// TIA Portal project "Project1" (V17)

(* hardware
DEVICE "S7-1200 station_1"  S7-1200 Station
   slot 0: "Rack_0"  S7-1200 Rack  Rack  V1.0
   slot 1: "PLC_1"  CPU 1215C AC/DC/Rly  6ES7 215-1BG40-0XB0  V4.5
*)

// ===== PLC "PLC_1"  CPU 1215C AC/DC/Rly =====

VAR_GLOBAL   // PLC tag table "input"
   "start" AT %I0.0 : Bool;
   "stop" AT %I0.1 : Bool;
   "cảm biến 1" AT %I0.2 : Bool;
   "cảm biến 2" AT %I0.3 : Bool;
   "cảm biến 3" AT %I0.4 : Bool;
   "cảm biến 4" AT %I0.5 : Bool;
   "cảm biến 5" AT %I0.6 : Bool;
   "auto" AT %I0.7 : Bool;
   "manual" AT %I1.0 : Bool;
   "emc" AT %I1.1 : Bool;
   "process1" AT %I1.2 : Bool;
   "process2" AT %I1.3 : Bool;
   "process3" AT %I1.4 : Bool;
END_VAR

VAR_GLOBAL   // PLC tag table "bit trung gian"
   "Tag_3" AT %M0.0 : Bool;
   "cam bien 1" AT %M0.1 : Bool;
   "hàng đỏ" AT %M1.0 : Bool;
   "hàng xanh lá" AT %M1.1 : Bool;
   "hàng xanh dương" AT %M1.2 : Bool;
   "hàng NG" AT %M1.3 : Bool;
   "cam bien 2" AT %M0.2 : Bool;
   "cảm bien 3" AT %M0.3 : Bool;
   "cam bien 4" AT %M0.4 : Bool;
   "cam bien 5" AT %M0.5 : Bool;
   "bit nho hang NG" AT %M0.6 : Bool;
   "bit nho van day 1" AT %M2.0 : Bool;
   "bit nho van day 2" AT %M2.1 : Bool;
   "Tag_4" AT %M2.2 : Bool;
   "Tag_5" AT %M2.3 : Bool;
   "bit nho van SP do" AT %M2.5 : Bool;
   "bit nho van SP xanh la" AT %M2.6 : Bool;
   "bit nho van sp xanh duong" AT %M2.7 : Bool;
   "bit nho van SP do 2" AT %M2.4 : Bool;
   "reset" AT %M3.0 : Bool;
   "bit nho bang tai" AT %M4.0 : Bool;
   "bit nho van xoay" AT %M4.1 : Bool;
   "bit nho van kep" AT %M4.2 : Bool;
   "bit nho van SP do 3" AT %M4.3 : Bool;
   "bit nho van xanh la 2" AT %M4.4 : Bool;
END_VAR

VAR_GLOBAL   // PLC tag table "bit output"
   "băng tải" AT %Q0.0 : Bool;
   "van sp đỏ" AT %Q0.1 : Bool;
   "Đèn xanh" AT %Q0.7 : Bool;
   "Đèn đỏ" AT %Q1.0 : Bool;
   "van xoay" AT %Q0.4 : Bool;
   "van đẩy tay gắp" AT %Q0.5 : Bool;
   "van kẹp tay gắp" AT %Q0.6 : Bool;
   "van sp xanh lá" AT %Q0.2 : Bool;
   "van sp xanh dương" AT %Q0.3 : Bool;
   "Đèn vàng" AT %Q1.1 : Bool;
END_VAR

DATA_BLOCK "DB1"   // DB1
{ S7_Optimized_Access := 'TRUE' }
VERSION : 0.1
   VAR
      disconnect : Bool;
      connect : TCON_IP_v4;
      error : Bool;
      h_reg : Array[0..50] of Int;
      status : Word;
   END_VAR
BEGIN
   connect.InterfaceId := 64;
   connect.ID := 1;
   connect.ConnectionType := 11;
   connect.LocalPort := 502;
   h_reg[16] := 0;
END_DATA_BLOCK

// folder: System blocks/Program resources

DATA_BLOCK "counter start"   // DB3
{ S7_Optimized_Access := 'TRUE' }
AUTHOR : Simatic
FAMILY : IEC
NAME : CNTR
VERSION : 1.0
// stored: InstanceOfName IEC_COUNTER
"IEC_COUNTER"
BEGIN
END_DATA_BLOCK

DATA_BLOCK "counter stop"   // DB4
{ S7_Optimized_Access := 'TRUE' }
AUTHOR : Simatic
FAMILY : IEC
NAME : CNTR
VERSION : 1.0
// stored: InstanceOfName IEC_COUNTER
"IEC_COUNTER"
BEGIN
END_DATA_BLOCK

DATA_BLOCK "T1"   // DB5
{ S7_Optimized_Access := 'TRUE' }
AUTHOR : Simatic
FAMILY : IEC
NAME : IEC_TMR
VERSION : 1.0
// stored: InstanceOfName IEC_TIMER
"IEC_TIMER"
BEGIN
END_DATA_BLOCK

DATA_BLOCK "timer hang xanh duong"   // DB6
{ S7_Optimized_Access := 'TRUE' }
AUTHOR : Simatic
FAMILY : IEC
NAME : IEC_TMR
VERSION : 1.0
// stored: InstanceOfName IEC_TIMER
"IEC_TIMER"
BEGIN
END_DATA_BLOCK

DATA_BLOCK "Counter dem hang xanh duong"   // DB7
{ S7_Optimized_Access := 'TRUE' }
AUTHOR : Simatic
FAMILY : IEC
NAME : CNTR
VERSION : 1.0
// stored: InstanceOfName IEC_COUNTER
"IEC_COUNTER"
BEGIN
END_DATA_BLOCK

DATA_BLOCK "xanh duong"   // DB8
{ S7_Optimized_Access := 'TRUE' }
AUTHOR : Simatic
FAMILY : IEC
NAME : CNTR
VERSION : 1.0
// stored: InstanceOfName IEC_COUNTER
"IEC_COUNTER"
BEGIN
END_DATA_BLOCK

DATA_BLOCK "đỏ"   // DB9
{ S7_Optimized_Access := 'TRUE' }
AUTHOR : Simatic
FAMILY : IEC
NAME : CNTR
VERSION : 1.0
// stored: InstanceOfName IEC_COUNTER
"IEC_COUNTER"
BEGIN
END_DATA_BLOCK

DATA_BLOCK "Timer hang do"   // DB10
{ S7_Optimized_Access := 'TRUE' }
AUTHOR : Simatic
FAMILY : IEC
NAME : IEC_TMR
VERSION : 1.0
// stored: InstanceOfName IEC_TIMER
"IEC_TIMER"
BEGIN
END_DATA_BLOCK

DATA_BLOCK "Counter dem hang do"   // DB11
{ S7_Optimized_Access := 'TRUE' }
AUTHOR : Simatic
FAMILY : IEC
NAME : CNTR
VERSION : 1.0
// stored: InstanceOfName IEC_COUNTER
"IEC_COUNTER"
BEGIN
END_DATA_BLOCK

DATA_BLOCK "xanh la cay"   // DB12
{ S7_Optimized_Access := 'TRUE' }
AUTHOR : Simatic
FAMILY : IEC
NAME : CNTR
VERSION : 1.0
// stored: InstanceOfName IEC_COUNTER
"IEC_COUNTER"
BEGIN
END_DATA_BLOCK

DATA_BLOCK "Timer xanh la cay"   // DB13
{ S7_Optimized_Access := 'TRUE' }
AUTHOR : Simatic
FAMILY : IEC
NAME : IEC_TMR
VERSION : 1.0
// stored: InstanceOfName IEC_TIMER
"IEC_TIMER"
BEGIN
END_DATA_BLOCK

DATA_BLOCK "Counter dem xanh la cay"   // DB14
{ S7_Optimized_Access := 'TRUE' }
AUTHOR : Simatic
FAMILY : IEC
NAME : CNTR
VERSION : 1.0
// stored: InstanceOfName IEC_COUNTER
"IEC_COUNTER"
BEGIN
END_DATA_BLOCK

DATA_BLOCK "IEC_Counter_0_DB"   // DB15
{ S7_Optimized_Access := 'TRUE' }
AUTHOR : Simatic
FAMILY : IEC
NAME : CNTR
VERSION : 1.0
// stored: InstanceOfName IEC_COUNTER
"IEC_COUNTER"
BEGIN
END_DATA_BLOCK

DATA_BLOCK "bao full do"   // DB16
{ S7_Optimized_Access := 'TRUE' }
AUTHOR : Simatic
FAMILY : IEC
NAME : CNTR
VERSION : 1.0
// stored: InstanceOfName IEC_COUNTER
"IEC_COUNTER"
BEGIN
END_DATA_BLOCK

DATA_BLOCK "bao full xanh la"   // DB17
{ S7_Optimized_Access := 'TRUE' }
AUTHOR : Simatic
FAMILY : IEC
NAME : CNTR
VERSION : 1.0
// stored: InstanceOfName IEC_COUNTER
"IEC_COUNTER"
BEGIN
END_DATA_BLOCK

DATA_BLOCK "bao ful xanh duong"   // DB18
{ S7_Optimized_Access := 'TRUE' }
AUTHOR : Simatic
FAMILY : IEC
NAME : CNTR
VERSION : 1.0
// stored: InstanceOfName IEC_COUNTER
"IEC_COUNTER"
BEGIN
END_DATA_BLOCK

DATA_BLOCK "hang NG"   // DB19
{ S7_Optimized_Access := 'TRUE' }
AUTHOR : Simatic
FAMILY : IEC
NAME : CNTR
VERSION : 1.0
// stored: InstanceOfName IEC_COUNTER
"IEC_COUNTER"
BEGIN
END_DATA_BLOCK

DATA_BLOCK "counter dem hang NG"   // DB20
{ S7_Optimized_Access := 'TRUE' }
AUTHOR : Simatic
FAMILY : IEC
NAME : CNTR
VERSION : 1.0
// stored: InstanceOfName IEC_COUNTER
"IEC_COUNTER"
BEGIN
END_DATA_BLOCK

DATA_BLOCK "bao full NG"   // DB21
{ S7_Optimized_Access := 'TRUE' }
AUTHOR : Simatic
FAMILY : IEC
NAME : CNTR
VERSION : 1.0
// stored: InstanceOfName IEC_COUNTER
"IEC_COUNTER"
BEGIN
END_DATA_BLOCK

DATA_BLOCK "counter cb 1"   // DB22
{ S7_Optimized_Access := 'TRUE' }
AUTHOR : Simatic
FAMILY : IEC
NAME : CNTR
VERSION : 1.0
// stored: InstanceOfName IEC_COUNTER
"IEC_COUNTER"
BEGIN
END_DATA_BLOCK

DATA_BLOCK "T2"   // DB23
{ S7_Optimized_Access := 'TRUE' }
AUTHOR : Simatic
FAMILY : IEC
NAME : IEC_TMR
VERSION : 1.0
// stored: InstanceOfName IEC_TIMER
"IEC_TIMER"
BEGIN
END_DATA_BLOCK

DATA_BLOCK "chay bang tai"   // DB24
{ S7_Optimized_Access := 'TRUE' }
AUTHOR : Simatic
FAMILY : IEC
NAME : CNTR
VERSION : 1.0
// stored: InstanceOfName IEC_COUNTER
"IEC_COUNTER"
BEGIN
END_DATA_BLOCK

DATA_BLOCK "IEC_Counter_0_DB_1"   // DB25
{ S7_Optimized_Access := 'TRUE' }
AUTHOR : Simatic
FAMILY : IEC
NAME : CNTR
VERSION : 1.0
// stored: InstanceOfName IEC_COUNTER
"IEC_COUNTER"
BEGIN
END_DATA_BLOCK

DATA_BLOCK "IEC_Counter_0_DB_2"   // DB26
{ S7_Optimized_Access := 'TRUE' }
AUTHOR : Simatic
FAMILY : IEC
NAME : CNTR
VERSION : 1.0
// stored: InstanceOfName IEC_COUNTER
"IEC_COUNTER"
BEGIN
END_DATA_BLOCK

DATA_BLOCK "IEC_Counter_0_DB_3"   // DB27
{ S7_Optimized_Access := 'TRUE' }
AUTHOR : Simatic
FAMILY : IEC
NAME : CNTR
VERSION : 1.0
// stored: InstanceOfName IEC_COUNTER
"IEC_COUNTER"
BEGIN
END_DATA_BLOCK

// folder: (top level)

FUNCTION "ouput" : Void   // FC1, LAD
{ S7_Optimized_Access := 'TRUE' }
VERSION : 0.1
BEGIN

REGION Network 1
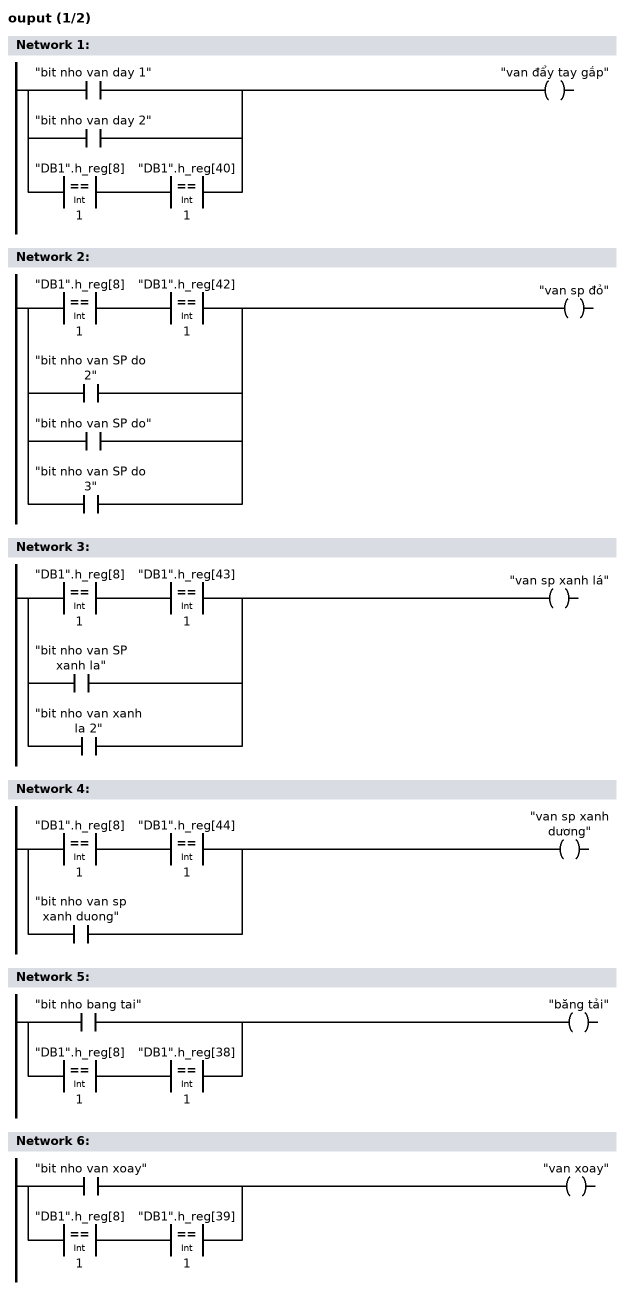
   RUNG wire#powerrail
      Contact( "bit nho van day 1" )
      wire#w1
      Coil( "van đẩy tay gắp" )
   END_RUNG
   RUNG wire#powerrail
      Contact( "bit nho van day 2" )
   END_RUNG wire#w1
   RUNG wire#powerrail
      { S7_Templates := "SrcType := Int" } EQ_Contact(in1 := "DB1".h_reg[8], in2 := 1)
      { S7_Templates := "SrcType := Int" } EQ_Contact(in1 := "DB1".h_reg[40], in2 := 1)
   END_RUNG wire#w1
   // the same network as SCL:
   "van đẩy tay gắp" := "bit nho van day 1" OR "bit nho van day 2" OR (("DB1".h_reg[8] = 1) AND ("DB1".h_reg[40] = 1));
END_REGION

REGION Network 2
   RUNG wire#powerrail
      { S7_Templates := "SrcType := Int" } EQ_Contact(in1 := "DB1".h_reg[8], in2 := 1)
      { S7_Templates := "SrcType := Int" } EQ_Contact(in1 := "DB1".h_reg[42], in2 := 1)
      wire#w1
      Coil( "van sp đỏ" )
   END_RUNG
   RUNG wire#powerrail
      Contact( "bit nho van SP do 2" )
   END_RUNG wire#w1
   RUNG wire#powerrail
      Contact( "bit nho van SP do" )
   END_RUNG wire#w1
   RUNG wire#powerrail
      Contact( "bit nho van SP do 3" )
   END_RUNG wire#w1
   // the same network as SCL:
   "van sp đỏ" := (("DB1".h_reg[8] = 1) AND ("DB1".h_reg[42] = 1)) OR "bit nho van SP do 2" OR "bit nho van SP do" OR "bit nho van SP do 3";
END_REGION

REGION Network 3
   RUNG wire#powerrail
      { S7_Templates := "SrcType := Int" } EQ_Contact(in1 := "DB1".h_reg[8], in2 := 1)
      { S7_Templates := "SrcType := Int" } EQ_Contact(in1 := "DB1".h_reg[43], in2 := 1)
      wire#w1
      Coil( "van sp xanh lá" )
   END_RUNG
   RUNG wire#powerrail
      Contact( "bit nho van SP xanh la" )
   END_RUNG wire#w1
   RUNG wire#powerrail
      Contact( "bit nho van xanh la 2" )
   END_RUNG wire#w1
   // the same network as SCL:
   "van sp xanh lá" := (("DB1".h_reg[8] = 1) AND ("DB1".h_reg[43] = 1)) OR "bit nho van SP xanh la" OR "bit nho van xanh la 2";
END_REGION

REGION Network 4
   RUNG wire#powerrail
      { S7_Templates := "SrcType := Int" } EQ_Contact(in1 := "DB1".h_reg[8], in2 := 1)
      { S7_Templates := "SrcType := Int" } EQ_Contact(in1 := "DB1".h_reg[44], in2 := 1)
      wire#w1
      Coil( "van sp xanh dương" )
   END_RUNG
   RUNG wire#powerrail
      Contact( "bit nho van sp xanh duong" )
   END_RUNG wire#w1
   // the same network as SCL:
   "van sp xanh dương" := (("DB1".h_reg[8] = 1) AND ("DB1".h_reg[44] = 1)) OR "bit nho van sp xanh duong";
END_REGION

REGION Network 5
   RUNG wire#powerrail
      Contact( "bit nho bang tai" )
      wire#w1
      Coil( "băng tải" )
   END_RUNG
   RUNG wire#powerrail
      { S7_Templates := "SrcType := Int" } EQ_Contact(in1 := "DB1".h_reg[8], in2 := 1)
      { S7_Templates := "SrcType := Int" } EQ_Contact(in1 := "DB1".h_reg[38], in2 := 1)
   END_RUNG wire#w1
   // the same network as SCL:
   "băng tải" := "bit nho bang tai" OR (("DB1".h_reg[8] = 1) AND ("DB1".h_reg[38] = 1));
END_REGION

REGION Network 6
   RUNG wire#powerrail
      Contact( "bit nho van xoay" )
      wire#w1
      Coil( "van xoay" )
   END_RUNG
   RUNG wire#powerrail
      { S7_Templates := "SrcType := Int" } EQ_Contact(in1 := "DB1".h_reg[8], in2 := 1)
      { S7_Templates := "SrcType := Int" } EQ_Contact(in1 := "DB1".h_reg[39], in2 := 1)
   END_RUNG wire#w1
   // the same network as SCL:
   "van xoay" := "bit nho van xoay" OR (("DB1".h_reg[8] = 1) AND ("DB1".h_reg[39] = 1));
END_REGION

REGION Network 7
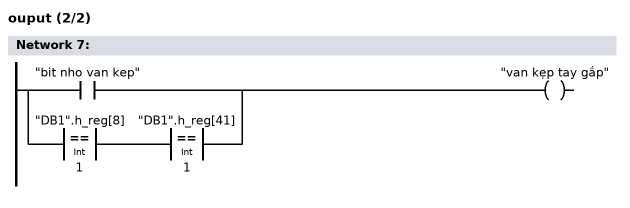
   RUNG wire#powerrail
      Contact( "bit nho van kep" )
      wire#w1
      Coil( "van kẹp tay gắp" )
   END_RUNG
   RUNG wire#powerrail
      { S7_Templates := "SrcType := Int" } EQ_Contact(in1 := "DB1".h_reg[8], in2 := 1)
      { S7_Templates := "SrcType := Int" } EQ_Contact(in1 := "DB1".h_reg[41], in2 := 1)
   END_RUNG wire#w1
   // the same network as SCL:
   "van kẹp tay gắp" := "bit nho van kep" OR (("DB1".h_reg[8] = 1) AND ("DB1".h_reg[41] = 1));
END_REGION
END_FUNCTION

FUNCTION "send signal to Python" : Void   // FC2, LAD
{ S7_Optimized_Access := 'TRUE' }
VERSION : 0.1
BEGIN

REGION Network 1
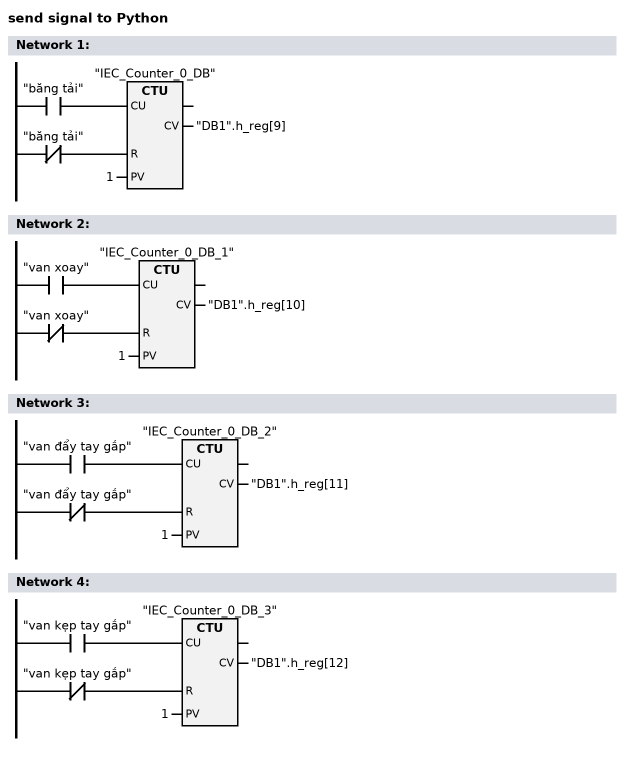
   "IEC_Counter_0_DB".CTU(CU := "băng tải", R := NOT "băng tải", PV := 1, CV => "DB1".h_reg[9]);
END_REGION

REGION Network 2
   "IEC_Counter_0_DB_1".CTU(CU := "van xoay", R := NOT "van xoay", PV := 1, CV => "DB1".h_reg[10]);
END_REGION

REGION Network 3
   "IEC_Counter_0_DB_2".CTU(CU := "van đẩy tay gắp", R := NOT "van đẩy tay gắp", PV := 1, CV => "DB1".h_reg[11]);
END_REGION

REGION Network 4
   "IEC_Counter_0_DB_3".CTU(CU := "van kẹp tay gắp", R := NOT "van kẹp tay gắp", PV := 1, CV => "DB1".h_reg[12]);
END_REGION
END_FUNCTION

FUNCTION "Red" : Void   // FC3, LAD
{ S7_Optimized_Access := 'TRUE' }
VERSION : 0.1
BEGIN

REGION Network 1
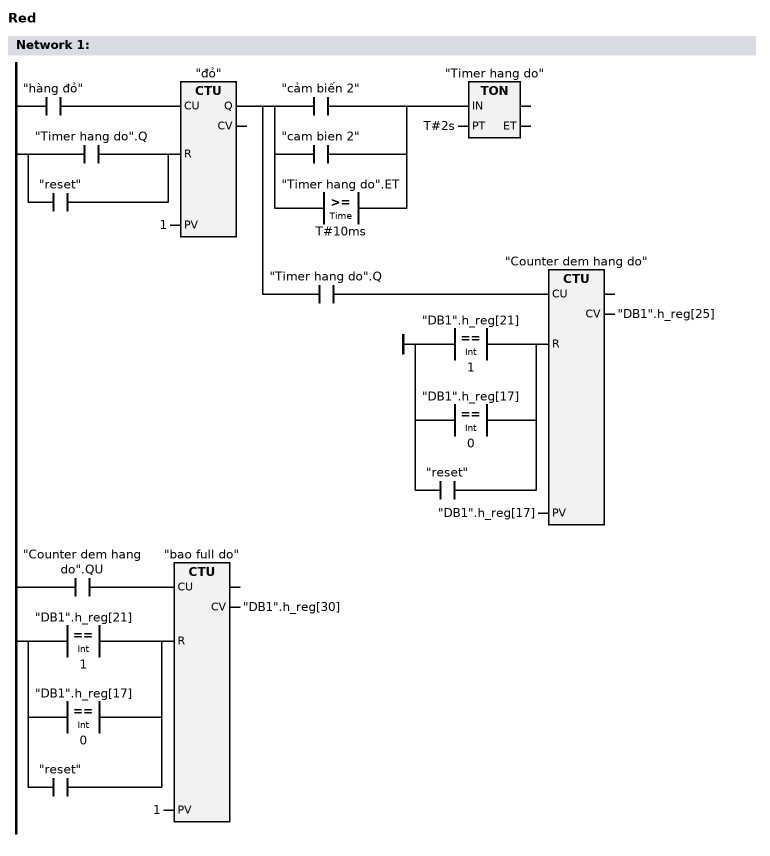
   "đỏ".CTU(CU := "hàng đỏ", R := "Timer hang do".Q OR "reset", PV := 1);
   "Timer hang do".TON(IN := "đỏ".Q AND ("cảm biến 2" OR "cam bien 2" OR ("Timer hang do".ET >= T#10ms)),
                       PT := T#2s);
   "Counter dem hang do".CTU(CU := "đỏ".Q AND "Timer hang do".Q,
                           R := ("DB1".h_reg[21] = 1) OR ("DB1".h_reg[17] = 0) OR "reset",
                           PV := "DB1".h_reg[17],
                           CV => "DB1".h_reg[25]);
   "bao full do".CTU(CU := "Counter dem hang do".QU,
                     R := ("DB1".h_reg[21] = 1) OR ("DB1".h_reg[17] = 0) OR "reset",
                     PV := 1,
                     CV => "DB1".h_reg[30]);
END_REGION
END_FUNCTION

FUNCTION "Green" : Void   // FC4, LAD
{ S7_Optimized_Access := 'TRUE' }
VERSION : 0.1
BEGIN

REGION Network 1
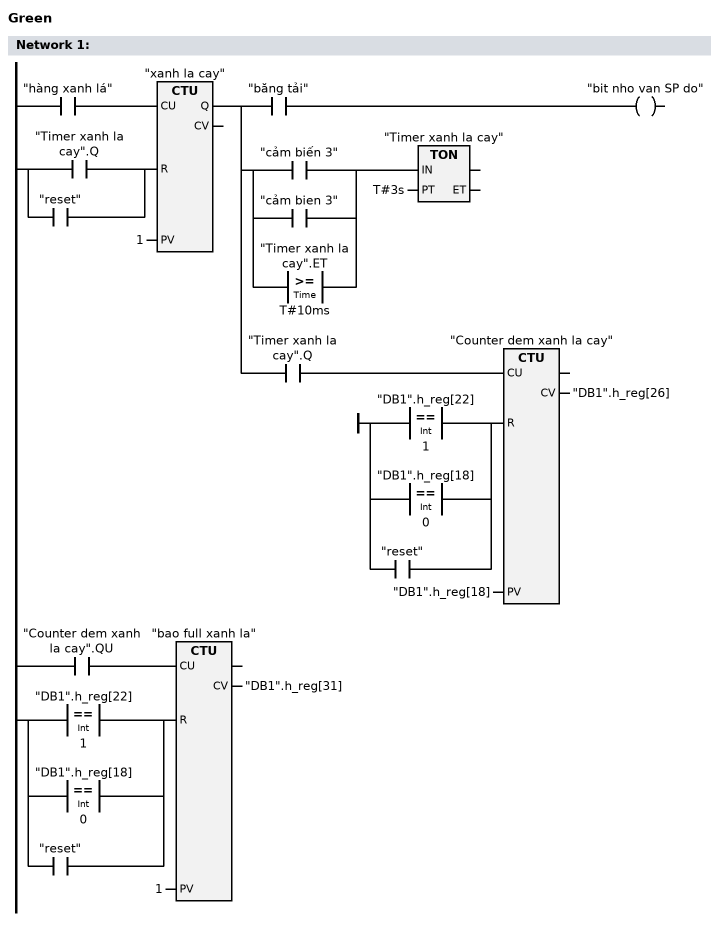
   "xanh la cay".CTU(CU := "hàng xanh lá", R := "Timer xanh la cay".Q OR "reset", PV := 1);
   "bit nho van SP do" := "xanh la cay".Q AND "băng tải";
   "Timer xanh la cay".TON(IN := "xanh la cay".Q AND ("cảm biến 3" OR "cảm bien 3" OR ("Timer xanh la cay".ET >= T#10ms)),
                           PT := T#3s);
   "Counter dem xanh la cay".CTU(CU := "xanh la cay".Q AND "Timer xanh la cay".Q,
                           R := ("DB1".h_reg[22] = 1) OR ("DB1".h_reg[18] = 0) OR "reset",
                           PV := "DB1".h_reg[18],
                           CV => "DB1".h_reg[26]);
   "bao full xanh la".CTU(CU := "Counter dem xanh la cay".QU,
                          R := ("DB1".h_reg[22] = 1) OR ("DB1".h_reg[18] = 0) OR "reset",
                          PV := 1,
                          CV => "DB1".h_reg[31]);
END_REGION
END_FUNCTION

FUNCTION "Blue" : Void   // FC5, LAD
{ S7_Optimized_Access := 'TRUE' }
VERSION : 0.1
BEGIN

REGION Network 1
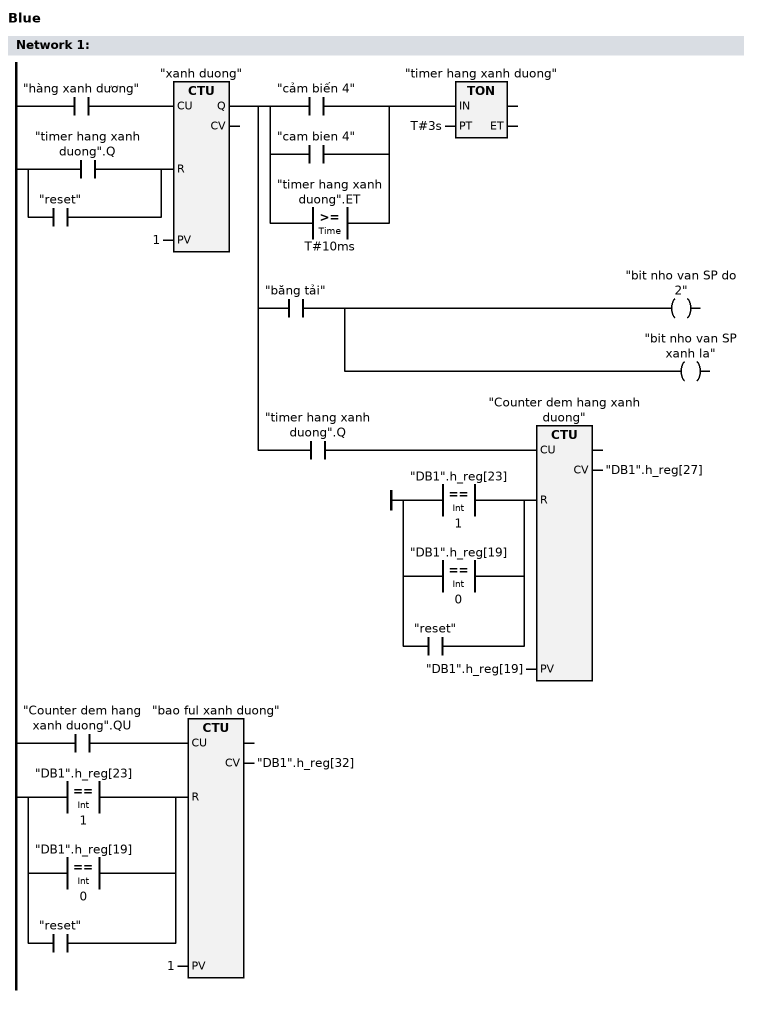
   "xanh duong".CTU(CU := "hàng xanh dương", R := "timer hang xanh duong".Q OR "reset", PV := 1);
   "timer hang xanh duong".TON(IN := "xanh duong".Q AND ("cảm biến 4" OR "cam bien 4" OR ("timer hang xanh duong".ET >= T#10ms)),
                           PT := T#3s);
   "bit nho van SP do 2" := "xanh duong".Q AND "băng tải";
   "bit nho van SP xanh la" := "bit nho van SP do 2";
   "Counter dem hang xanh duong".CTU(CU := "xanh duong".Q AND "timer hang xanh duong".Q,
                           R := ("DB1".h_reg[23] = 1) OR ("DB1".h_reg[19] = 0) OR "reset",
                           PV := "DB1".h_reg[19],
                           CV => "DB1".h_reg[27]);
   "bao ful xanh duong".CTU(CU := "Counter dem hang xanh duong".QU,
                           R := ("DB1".h_reg[23] = 1) OR ("DB1".h_reg[19] = 0) OR "reset",
                           PV := 1,
                           CV => "DB1".h_reg[32]);
END_REGION
END_FUNCTION

FUNCTION "NG" : Void   // FC6, LAD
{ S7_Optimized_Access := 'TRUE' }
VERSION : 0.1
BEGIN

REGION Network 1
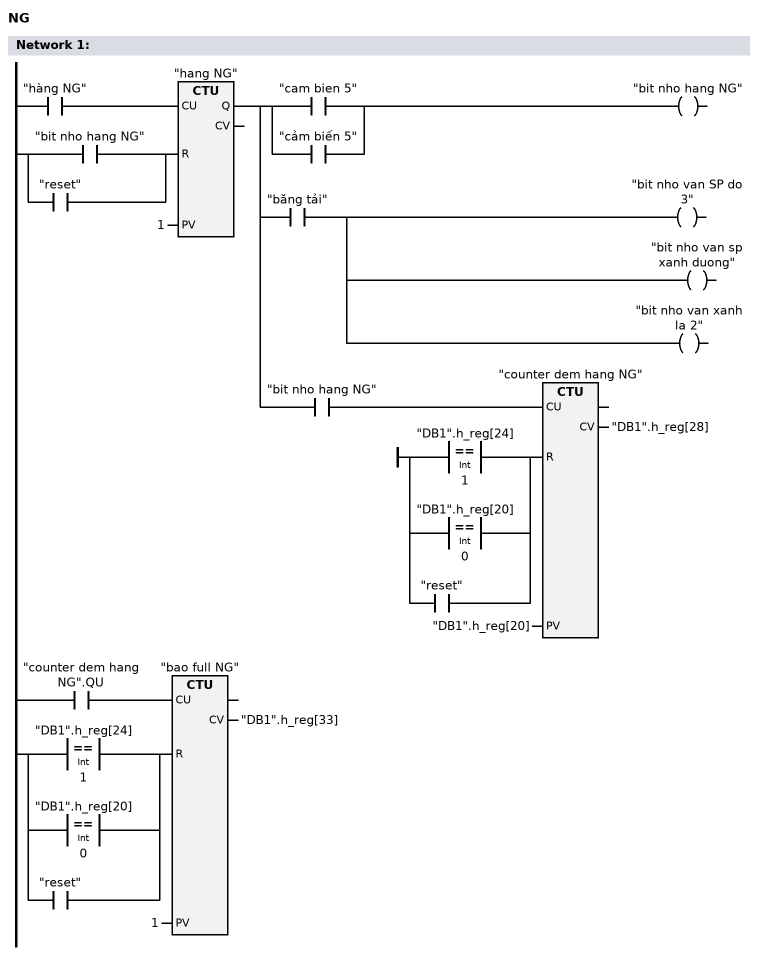
   "hang NG".CTU(CU := "hàng NG", R := "bit nho hang NG" OR "reset", PV := 1);
   "bit nho hang NG" := "hang NG".Q AND ("cam bien 5" OR "cảm biến 5");
   "bit nho van SP do 3" := "hang NG".Q AND "băng tải";
   "bit nho van sp xanh duong" := "bit nho van SP do 3";
   "bit nho van xanh la 2" := "bit nho van SP do 3";
   "counter dem hang NG".CTU(CU := "hang NG".Q AND "bit nho hang NG",
                           R := ("DB1".h_reg[24] = 1) OR ("DB1".h_reg[20] = 0) OR "reset",
                           PV := "DB1".h_reg[20],
                           CV => "DB1".h_reg[28]);
   "bao full NG".CTU(CU := "counter dem hang NG".QU,
                     R := ("DB1".h_reg[24] = 1) OR ("DB1".h_reg[20] = 0) OR "reset",
                     PV := 1,
                     CV => "DB1".h_reg[33]);
END_REGION
END_FUNCTION

ORGANIZATION_BLOCK "Main"   // OB1, LAD, ProgramCycle
TITLE = "Main Program Sweep (Cycle)"
{ S7_Optimized_Access := 'TRUE' }
VERSION : 0.1
   VAR_INPUT
      Initial_Call : Bool;   // Initial call of this OB
      Remanence : Bool;   // =True, if remanent data are available
   END_VAR
   VAR_TEMP   // added for the SCL form of the ladder/FBD networks
      _w1 : Bool;
   END_VAR
BEGIN

REGION Network 1
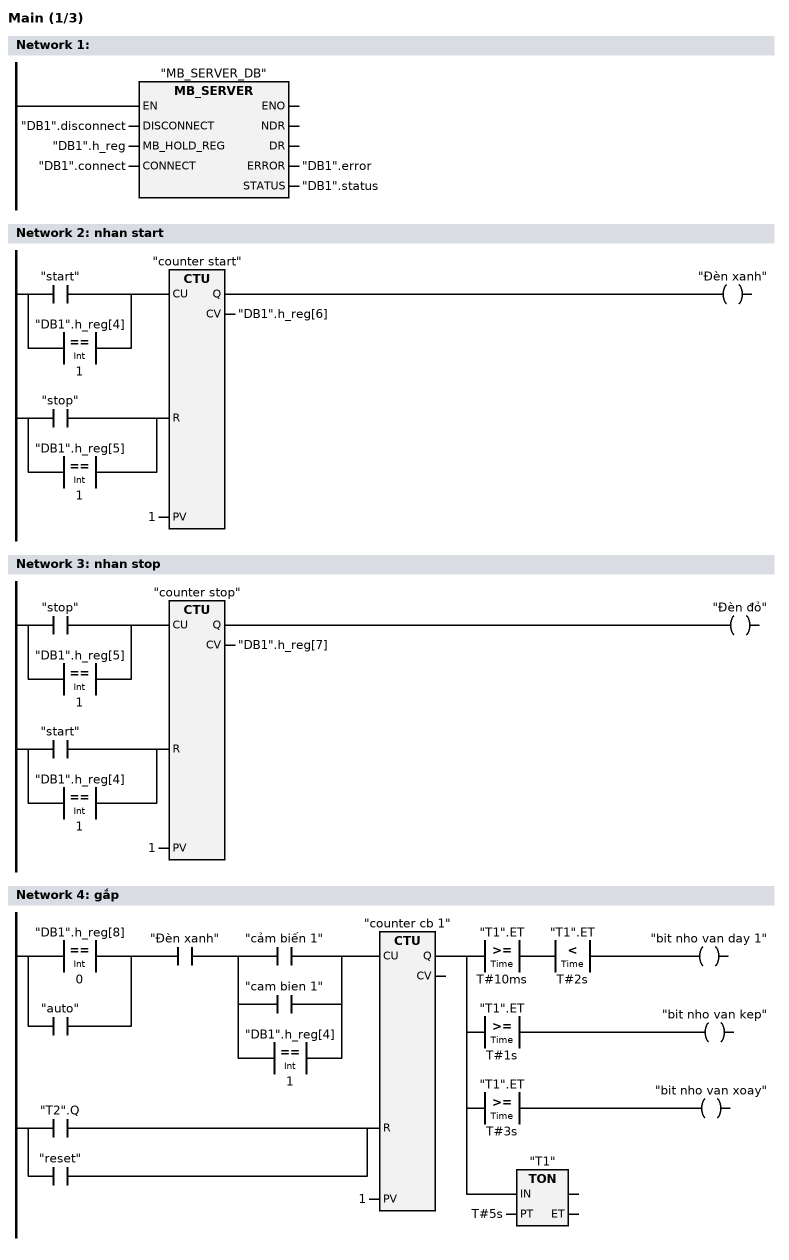
   "MB_SERVER_DB"(DISCONNECT := "DB1".disconnect,   // MB_SERVER
                  MB_HOLD_REG := "DB1".h_reg,
                  CONNECT := "DB1".connect,
                  ERROR => "DB1".error,
                  STATUS => "DB1".status);
END_REGION

REGION Network 2: nhan start
   "counter start".CTU(CU := "start" OR ("DB1".h_reg[4] = 1),
                       R := "stop" OR ("DB1".h_reg[5] = 1),
                       PV := 1,
                       CV => "DB1".h_reg[6]);
   "Đèn xanh" := "counter start".Q;
END_REGION

REGION Network 3: nhan stop
   "counter stop".CTU(CU := "stop" OR ("DB1".h_reg[5] = 1),
                      R := "start" OR ("DB1".h_reg[4] = 1),
                      PV := 1,
                      CV => "DB1".h_reg[7]);
   "Đèn đỏ" := "counter stop".Q;
END_REGION

REGION Network 4: gắp
   "counter cb 1".CTU(CU := (("DB1".h_reg[8] = 0) OR "auto") AND "Đèn xanh" AND ("cảm biến 1" OR "cam bien 1" OR ("DB1".h_reg[4] = 1)),
                      R := "T2".Q OR "reset",
                      PV := 1);
   "bit nho van day 1" := "counter cb 1".Q AND ("T1".ET >= T#10ms) AND ("T1".ET < T#2s);
   "bit nho van kep" := "counter cb 1".Q AND ("T1".ET >= T#1s);
   "bit nho van xoay" := "counter cb 1".Q AND ("T1".ET >= T#3s);
   "T1".TON(IN := "counter cb 1".Q, PT := T#5s);
END_REGION

REGION Network 5: dung de nhan dien hang
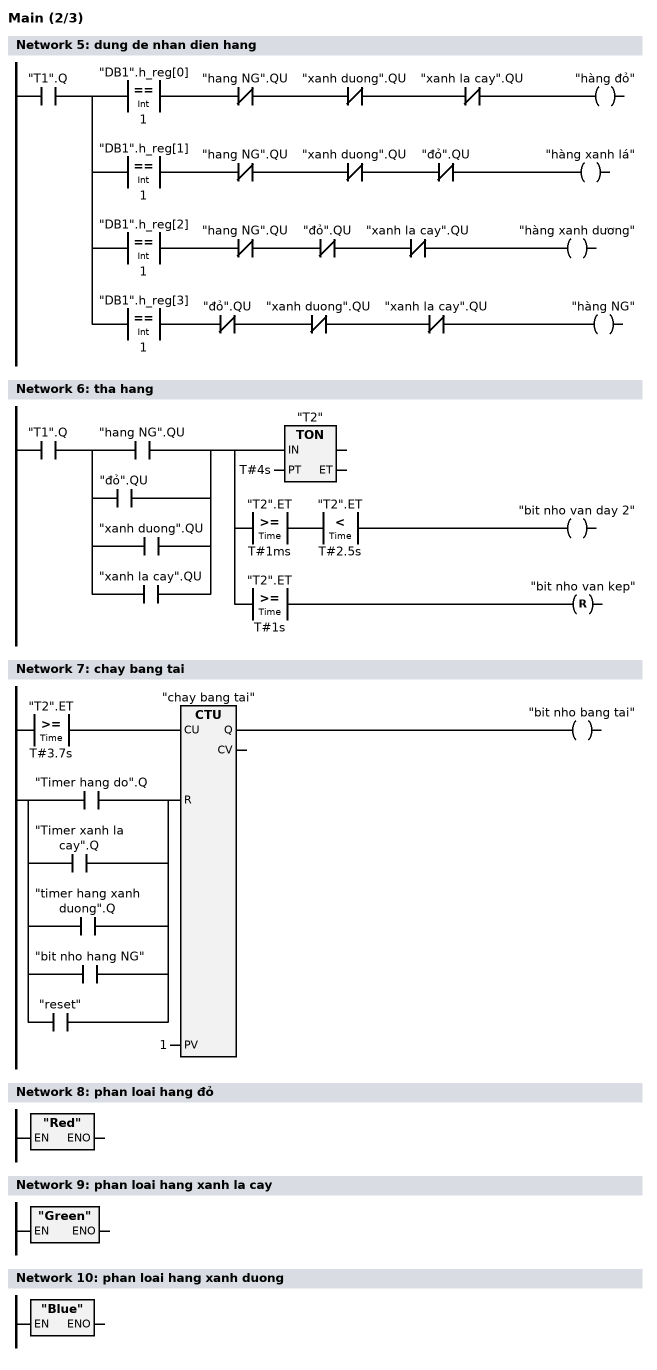
   RUNG wire#powerrail
      Contact( "T1".Q )
      wire#w1
      { S7_Templates := "SrcType := Int" } EQ_Contact(in1 := "DB1".h_reg[0], in2 := 1)
      I_Contact( "hang NG".QU )
      I_Contact( "xanh duong".QU )
      I_Contact( "xanh la cay".QU )
      Coil( "hàng đỏ" )
   END_RUNG
   RUNG wire#w1
      { S7_Templates := "SrcType := Int" } EQ_Contact(in1 := "DB1".h_reg[1], in2 := 1)
      I_Contact( "hang NG".QU )
      I_Contact( "xanh duong".QU )
      I_Contact( "đỏ".QU )
      Coil( "hàng xanh lá" )
   END_RUNG
   RUNG wire#w1
      { S7_Templates := "SrcType := Int" } EQ_Contact(in1 := "DB1".h_reg[2], in2 := 1)
      I_Contact( "hang NG".QU )
      I_Contact( "đỏ".QU )
      I_Contact( "xanh la cay".QU )
      Coil( "hàng xanh dương" )
   END_RUNG
   RUNG wire#w1
      { S7_Templates := "SrcType := Int" } EQ_Contact(in1 := "DB1".h_reg[3], in2 := 1)
      I_Contact( "đỏ".QU )
      I_Contact( "xanh duong".QU )
      I_Contact( "xanh la cay".QU )
      Coil( "hàng NG" )
   END_RUNG
   // the same network as SCL:
   "hàng đỏ" := "T1".Q AND ("DB1".h_reg[0] = 1) AND NOT "hang NG".QU AND NOT "xanh duong".QU AND NOT "xanh la cay".QU;
   "hàng xanh lá" := "T1".Q AND ("DB1".h_reg[1] = 1) AND NOT "hang NG".QU AND NOT "xanh duong".QU AND NOT "đỏ".QU;
   "hàng xanh dương" := "T1".Q AND ("DB1".h_reg[2] = 1) AND NOT "hang NG".QU AND NOT "đỏ".QU AND NOT "xanh la cay".QU;
   "hàng NG" := "T1".Q AND ("DB1".h_reg[3] = 1) AND NOT "đỏ".QU AND NOT "xanh duong".QU AND NOT "xanh la cay".QU;
END_REGION

REGION Network 6: tha hang
   #_w1 := "T1".Q AND ("hang NG".QU OR "đỏ".QU OR "xanh duong".QU OR "xanh la cay".QU);
   "T2".TON(IN := #_w1, PT := T#4s);
   "bit nho van day 2" := #_w1 AND ("T2".ET >= T#1ms) AND ("T2".ET < T#2.5s);
   IF #_w1 AND ("T2".ET >= T#1s) THEN "bit nho van kep" := FALSE; END_IF;
END_REGION

REGION Network 7: chay bang tai
   "chay bang tai".CTU(CU := "T2".ET >= T#3.7s,
                       R := "Timer hang do".Q OR "Timer xanh la cay".Q OR "timer hang xanh duong".Q OR "bit nho hang NG" OR "reset",
                       PV := 1);
   "bit nho bang tai" := "chay bang tai".Q;
END_REGION

REGION Network 8: phan loai hang đỏ
   RUNG wire#powerrail
      "Red"()
   END_RUNG
   // the same network as SCL:
   "Red"();
END_REGION

REGION Network 9: phan loai hang xanh la cay
   RUNG wire#powerrail
      "Green"()
   END_RUNG
   // the same network as SCL:
   "Green"();
END_REGION

REGION Network 10: phan loai hang xanh duong
   RUNG wire#powerrail
      "Blue"()
   END_RUNG
   // the same network as SCL:
   "Blue"();
END_REGION

REGION Network 11: phan loai hang NG
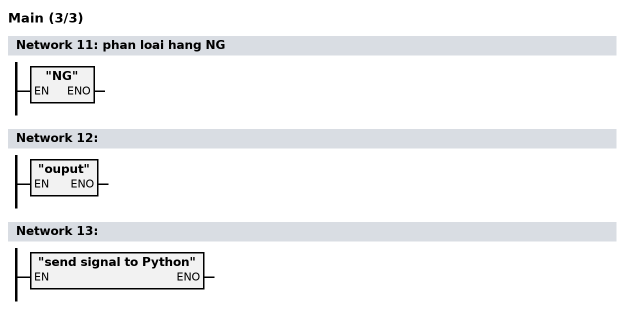
   RUNG wire#powerrail
      "NG"()
   END_RUNG
   // the same network as SCL:
   "NG"();
END_REGION

REGION Network 12
   RUNG wire#powerrail
      "ouput"()
   END_RUNG
   // the same network as SCL:
   "ouput"();
END_REGION

REGION Network 13
   RUNG wire#powerrail
      "send signal to Python"()
   END_RUNG
   // the same network as SCL:
   "send signal to Python"();
END_REGION
END_ORGANIZATION_BLOCK